// TIA Portal V21 export
// export: Created 2026-08-27T15:25:32.7339811Z, ExportSetting None, DisplayName Totally Integrated Automation Portal, DisplayVersion V21, DisplayName STEP 7 Professional, DisplayVersion V21, DisplayName STEP 7 Safety, DisplayVersion V21, DisplayName Tech WebApplication, DisplayVersion V21, DisplayName WinCC Basic/Comfort/Advanced, DisplayVersion V21
VAR_GLOBAL   // PLC tag table "TASK014_Acceptance_IO"
   StartButton AT %I0.0 : Bool;
   StopButton AT %I0.1 : Bool;
   ResetButton AT %I0.2 : Bool;
   EmergencyOk AT %I0.3 : Bool;
   AutoMode AT %I0.4 : Bool;
   PartSensor AT %I0.5 : Bool;
   MotorRun AT %Q0.0 : Bool;
   AlarmLamp AT %Q0.1 : Bool;
   ValveExtend AT %Q0.2 : Bool;
   ValveRetract AT %Q0.3 : Bool;
END_VAR
